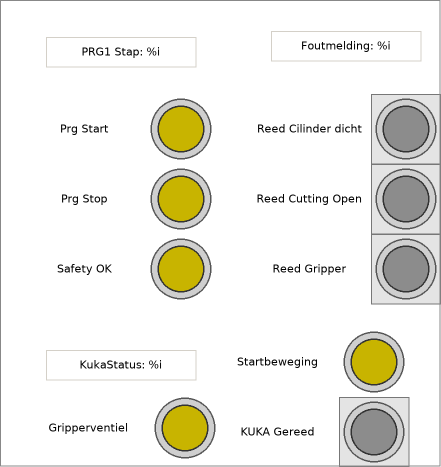
VISUALIZATION HMI  // 441x467
    Group (248,94 193x210)
        PushSwitch (123,0 70x70), variable: DB10_Alias.ix_reedCuttingtoolCilinderGesloten, behaviour: TOGGLE, style: Switch-PushSwitch-Gray
        Label (0,20 123x30), "Reed Cilinder dicht"
        PushSwitch (123,70 70x70), variable: DB10_Alias.ix_reedCuttingtoolCilinderOpen, behaviour: TOGGLE, style: Switch-PushSwitch-Gray
        Label (0,90 123x30), "Reed Cutting Open"
        PushSwitch (123,140 70x70), variable: DB10_Alias.ix_reedGripperCilinder1, behaviour: TAP, style: Switch-PushSwitch-Gray
        Label (0,160 123x30), "Reed Gripper"
    Textfield (46,37 150x30), "PRG1 Stap: %i", text variable: DB_PRG1.PRG1Stap
    Group (23,94 193x70)
        Label (0,20 123x30), "Prg Start"
        Lamp1 (123,0 70x70), variable: GVL.b_StartPRG, style: Lamp-Lamp1-Yellow
    Group (23,164 193x70)
        Label (0,20 123x30), "Prg Stop"
        Lamp1 (123,0 70x70), variable: GVL.b_StopPRG, style: Lamp-Lamp1-Yellow
    Group (23,234 193x70)
        Label (0,20 123x30), "Safety OK"
        Lamp1 (123,0 70x70), variable: GVL.safetyOK, style: Lamp-Lamp1-Yellow
    Textfield (271,31 150x30), "Foutmelding: %i", text variable: FC_PRG1.Foutcode
    Textfield (46,350 150x30), "KukaStatus: %i", text variable: GVL.i_KUKAStatus
    Group (216,327 193x70)
        Label (0,20 123x30), "Startbeweging"
        Lamp1 (123,0 70x70), variable: GVL.b_startBeweging, style: Lamp-Lamp1-Yellow
    PushSwitch (339,397 70x70), variable: DB10_Alias.ix_kukaGereed, behaviour: TOGGLE, style: Switch-PushSwitch-Gray
    Label (216,417 123x30), "KUKA Gereed"
    Label (27,413 123x30), "Gripperventiel"
    Lamp1 (150,393 70x70), variable: DB10_Alias.qx_ventielEen, style: Lamp-Lamp1-Yellow
END_VISUALIZATION

(* stored: Version 1.1.0.1, ProductVersion 3.1.4024.12
   Visu HMI: Id {c27db630-7a49-4b8e-9b22-a3e1c24688ec} *)
